Universal Robots PolyScope program: mqtt_base_v2.urp

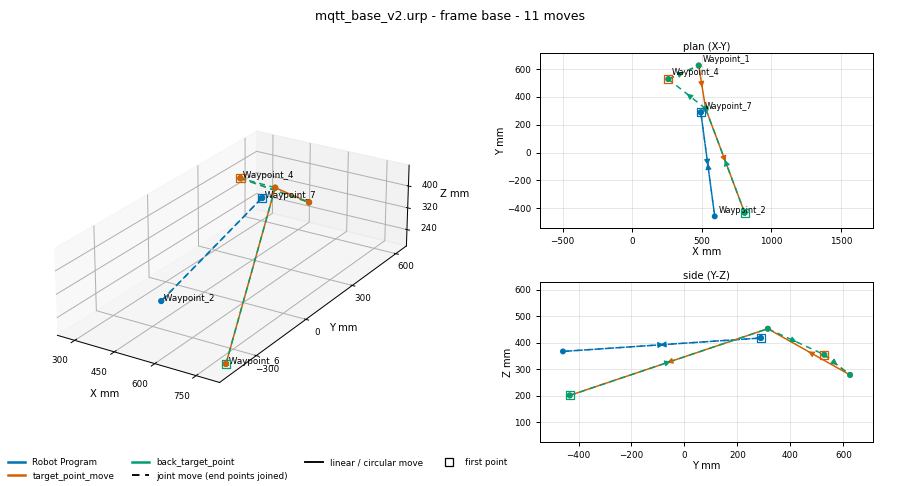
[picture p0: tool path of mqtt_base_v2.urp in frame base, 11 of 12 moves have a stored position in this frame; points joined in program order, loops and branches not executed]
Program mqtt base v2 (installation=default directory=/programs/usbdisk/new folder createdIn=5.13.0 lastSavedIn=5.13.0 robotSerialNumber=20205001820)
Calibrated DH parameters: a=[0.000063, -0.611934, -0.498535, 0.00003, -0.000005, 0]; d=[0.180864, 8.608021, 86.773068, -95.207056, 0.119988, 0.115697]; alpha=[1.571267, -0.001739, -0.002927, 1.571188, -1.571145, 0]; deltaTheta=[0, -0.024461, -0.486053, 0.510519, 0, 0]
InitVariablesNode variables(variable(name=distance, expression=p[0,0,0,0,0,0]), variable(name=freedrive, expression=0), variable(name=new_pos, expression=[0,0,0,0,0,0]), variable(name=order, expression=0), variable(name=program_loop, expression=0), variable(name=stop, expression=0), variable(name=target_point, expression=0), variable(name=topic_order, expression="robot"))
BeforeStart
  var_1 := mqtt_initialize_anonymous("192.168.4.1", 1883)
  var_2 := mqtt_connect()
  var_3 := mqtt_subscribe(topic_order)
Robot Program (runOnlyOnce=true)
  MoveJ speed 60 deg/s, acceleration 80 deg/s^2 (useActiveTCP=true) feature=Base
    Waypoint Waypoint_7: TCP in base x=492.803 y=288.649 z=418.324 mm, rx=2.6568 ry=-1.6608 rz=-0.0199 rad; joints [192.415, -98.238, 124.325, -115.253, -89.954, -13.481] deg
  Loop Forever
    Switch expression=order
      Case (caseValue=1)
        Wait Sleep waitTime=0.3
        Call target_point_move
        rst_mqtt := mqtt_publish(topic_order, " ", 1,  True )
        order := 6
      Case (caseValue=2)
        Wait Sleep waitTime=0.3
        Call back_target_point
        rst_mqtt := mqtt_publish(topic_order, " ", 1,  True )
        order := 6
      Case (caseValue=3)
        mqtt_send_fc := mqtt_publish("robot/return", order, 0,  False )
        distance := p[new_pos[0],new_pos[1],new_pos[2],new_pos[3],new_pos[4],new_pos[5]]
        Call move
        order := 0
        distance := p[0,0,0,0,0,0]
        rst_mqtt := mqtt_publish(topic_order, " ", 1,  True )
      Case (caseValue=4)
        MoveJ speed 60 deg/s, acceleration 80 deg/s^2 (useActiveTCP=true) feature=Base
          Waypoint Waypoint_2: TCP in base x=592.766 y=-458.734 z=367.679 mm, rx=-0.6196 ry=3.0445 rz=0.014 rad; joints [128.391, -78.663, 110.233, -122.029, -88.154, 15.462] deg
        Loop While (checkContinuously=true) expression=order==4
          Script file /programs/freedrive.script
            | freedrive_mode()
        Script file /programs/end_freedrive.script
          | end_freedrive_mode()
      Case (caseValue=6)
        MoveJ speed 60 deg/s, acceleration 80 deg/s^2 (useActiveTCP=true) feature=Base
          Waypoint Waypoint_3: TCP in base x=492.802 y=288.666 z=418.31 mm, rx=2.6568 ry=-1.6607 rz=-0.0199 rad; joints [192.417, -98.236, 124.324, -115.253, -89.956, -13.481] deg
        order := 0
      Case (caseValue=2147483647)
        Wait Sleep waitTime=0.5
Thread Thread_3 (runOnlyOnce=false)
  Wait Sleep waitTime=0.5
  If order==5
    Script: stopj(2)
SubProgram -> move
Thread Thread_1 (runOnlyOnce=false)
  Loop Forever
    Wait Sleep waitTime=0.5
    program_loop := mqtt_get_json_message(topic_order, "program_loop", program_loop)
    target_point := mqtt_get_json_message(topic_order, "target_point", target_point)
    freedrive := mqtt_get_json_message(topic_order, "freedrive", freedrive)
    new_pos := mqtt_get_json_message(topic_order, "new_pos", new_pos)
    stop := mqtt_get_json_message(topic_order, "stop", stop)
    order := mqtt_get_json_message(topic_order, "order", order)
SubProgram -> back_target_point
SubProgram -> target_point_move
SubProgram target_point_move (keepSynchronizedWithDisk=false)
  Wait Sleep waitTime=0.5
  MoveL speed 250 mm/s, acceleration 1200 mm/s^2 (useActiveTCP=true) feature=Base
    MoveDirectionNode (selectedDirection=ZPlus)
      Until DISTANCE (allowActions=false deceleration=3 distanceNodeType=STOP) Distance=0.2; motionParameters(blendRadius=0)
  Switch expression=target_point
    Case (caseValue=1)
      MoveJ speed 60 deg/s, acceleration 80 deg/s^2 (useActiveTCP=true) feature=Base
        Waypoint Waypoint_4: TCP in base x=259.212 y=527.898 z=355.358 mm, rx=-2.6848 ry=1.6264 rz=-0.0183 rad; joints [226.614, -92.85, 127.172, -124.624, -90.757, 19.087] deg
    Case (caseValue=2)
      MoveJ speed 60 deg/s, acceleration 80 deg/s^2 (useActiveTCP=true) feature=Base
        Waypoint Waypoint_1: TCP in base x=477.624 y=625.24 z=278.948 mm, rx=-2.6325 ry=1.6869 rz=0.0449 rad; joints [219.454, -70.395, 109.973, -129.892, -88.344, 14.805] deg
  URCap RG Grip (OnRobot, OnRobot A/S) dataModel(rg-target-force=40.0, rg-depth-compensation-enabled=true, rg-target-width=0.11)
  MoveL speed 250 mm/s, acceleration 1200 mm/s^2 (useActiveTCP=true) feature=Base
    MoveDirectionNode (selectedDirection=ZMinus toolParams=0.05, 1.2)
      Until TOOL_CONTACT_DETECTION (allowActions=false retraction=0.005 decelerationAcceleration=3 decelerationAngularAcceleration=34.906585)
    URCap RG Grip (OnRobot, OnRobot A/S) dataModel(rg-depth-compensation-enabled=true, rg-target-width=0.010199999999999999, workpiece-lost=false, payload-weight=0.5, rg-target-force=22.0, Variable(key=on_return, variable(name=on_return)))
    MoveDirectionNode (selectedDirection=ZPlus)
      Until DISTANCE (allowActions=false deceleration=3 distanceNodeType=STOP) Distance=0.3; motionParameters(blendRadius=0)
    Waypoint Waypoint_5: TCP in base x=527.445 y=314.854 z=453.36 mm, rx=2.6279 ry=-1.7134 rz=-0.0112 rad; joints [194.188, -95.358, 118.077, -112.277, -89.995, -9.507] deg
    Waypoint Waypoint_6: TCP in base x=807.912 y=-433.125 z=201.587 mm, rx=-0.6852 ry=3.024 rz=-0.0161 rad; joints [140.573, -55.8, 96.757, -132.886, -88.708, 25.083] deg
    MoveDirectionNode (selectedDirection=ZMinus toolParams=0.05, 1.2)
      Until TOOL_CONTACT_DETECTION (allowActions=false retraction=0.003 decelerationAcceleration=3 decelerationAngularAcceleration=34.906585)
    URCap RG Grip (OnRobot, OnRobot A/S) dataModel(rg-target-force=40.0, rg-depth-compensation-enabled=true, rg-target-width=0.11)
SubProgram back_target_point (keepSynchronizedWithDisk=false)
  If freedrive≠1
    MoveJ speed 60 deg/s, acceleration 80 deg/s^2 (useActiveTCP=true) feature=Base
      Waypoint Waypoint_6: TCP in base x=807.912 y=-433.125 z=201.587 mm, rx=-0.6852 ry=3.024 rz=-0.0161 rad; joints [140.573, -55.8, 96.757, -132.886, -88.708, 25.083] deg
  URCap RG Grip (OnRobot, OnRobot A/S) dataModel(rg-target-force=40.0, rg-depth-compensation-enabled=true, rg-target-width=0.11)
  MoveL speed 250 mm/s, acceleration 1200 mm/s^2 (useActiveTCP=true) feature=Base
    MoveDirectionNode (selectedDirection=ZMinus toolParams=0.05, 1.2)
      Until TOOL_CONTACT_DETECTION (allowActions=false retraction=0.003 decelerationAcceleration=3 decelerationAngularAcceleration=34.906585)
  URCap RG Grip (OnRobot, OnRobot A/S) dataModel(rg-target-force=40.0, rg-target-width=0.0085, rg-depth-compensation-enabled=true, Variable(key=on_return, variable=on_return))
  MoveL speed 250 mm/s, acceleration 1200 mm/s^2 (useActiveTCP=true) feature=Base
    MoveDirectionNode (selectedDirection=ZPlus)
      Until DISTANCE (allowActions=false deceleration=3 distanceNodeType=STOP) Distance=0.2; motionParameters(blendRadius=0)
  MoveJ speed 60 deg/s, acceleration 80 deg/s^2 (useActiveTCP=true) feature=Base
    Waypoint Waypoint_5: TCP in base x=527.445 y=314.854 z=453.36 mm, rx=2.6279 ry=-1.7134 rz=-0.0112 rad; joints [194.188, -95.358, 118.077, -112.277, -89.995, -9.507] deg
  Switch expression=target_point
    Case (caseValue=1)
      MoveJ speed 60 deg/s, acceleration 80 deg/s^2 (useActiveTCP=true) feature=Base
        Waypoint Waypoint_4: TCP in base x=259.212 y=527.898 z=355.358 mm, rx=-2.6848 ry=1.6264 rz=-0.0183 rad; joints [226.614, -92.85, 127.172, -124.624, -90.757, 19.087] deg
    Case (caseValue=2)
      MoveJ speed 60 deg/s, acceleration 80 deg/s^2 (useActiveTCP=true) feature=Base
        Waypoint Waypoint_10: TCP in base x=477.61 y=625.283 z=278.969 mm, rx=-2.6325 ry=1.6869 rz=0.0448 rad; joints [219.458, -70.394, 109.971, -129.895, -88.347, 14.807] deg
  MoveL speed 250 mm/s, acceleration 1200 mm/s^2 (useActiveTCP=true) feature=Base
    MoveDirectionNode (selectedDirection=ZMinus toolParams=0.05, 1.2)
      Until TOOL_CONTACT_DETECTION (allowActions=false retraction=0.003 decelerationAcceleration=3 decelerationAngularAcceleration=34.906585)
  URCap RG Grip (OnRobot, OnRobot A/S) dataModel(rg-target-force=40.0, rg-depth-compensation-enabled=true, rg-target-width=0.11)
SubProgram move (keepSynchronizedWithDisk=false)
  MoveL speed 250 mm/s, acceleration 1200 mm/s^2 (useActiveTCP=true) feature=Joint_6_name
    Waypoint Variable (Variable): variable(name=distance)
